// TIA Portal V20 export
TYPE "LWONIK_typeScrapBoxCommand"
// stored: Access Published
   STRUCT
      lock { ExternalWritable := 'False'} : Bool;
      unlock { ExternalWritable := 'False'} : Bool;
      reset { ExternalWritable := 'False'} : Bool;
   END_STRUCT;
END_TYPE
